FUNCTION_BLOCK TN_SC_WRITE_C
VAR
	FB_TN_SC_WRITE : TN_SC_WRITE;
END_VAR
VAR_INPUT
	Iin_Y : INT;
	Iin_X : INT;
	Iby_ATTR : BYTE;
	Ist_STRING : STRING;
	Iin_LENGTH : INT;
	Iin_OPTION : INT;
END_VAR
VAR_IN_OUT
	Xus_TN_SCREEN : us_TN_SCREEN;
END_VAR

(*
version 1.0		10. mai 2010
programmer		ks
tested by		ks

TN_SC_WRITE_C korrigiert die Textlänge und schreibt den Text an die angegebenen Koordinate
*)

(* Text ausgeben *)
FB_TN_SC_WRITE( Iin_Y := Iin_Y,
				Iin_X := Iin_X,
				Iby_ATTR := Iby_ATTR,
				Ist_STRING := FIX(str:=Ist_STRING,L:=Iin_LENGTH,C:=BYTE#32,M:=Iin_OPTION),
				Xus_TN_SCREEN := Xus_TN_SCREEN);

(* revision history
ks	10. mai. 2010	rev 1.0
	original version
*)

END_FUNCTION_BLOCK

(* stored: Version 1.1.0.1, ProductVersion 3.1.4024.9
   POU TN_SC_WRITE_C: Id {a46e4b68-3e91-4f58-8927-7cf0d0199213}, SpecialFunc None *)
